// Mitsubishi GX Works2 project: traffic signal with data   PLC: FX1N/FX1NC

PROGRAM MAIN
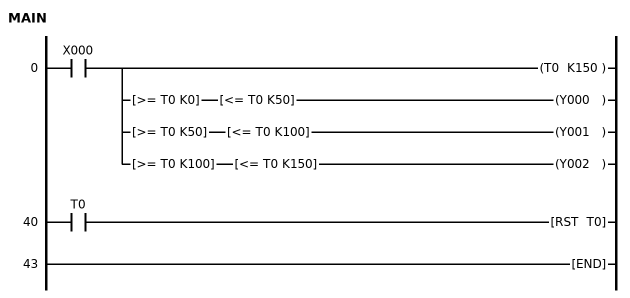
0     LD      X000
      OUT     T0 K150
      MPS
      AND>=   T0 K0
      AND<=   T0 K50
      OUT     Y000
      MRD
      AND>=   T0 K50
      AND<=   T0 K100
      OUT     Y001
      MPP
      AND>=   T0 K100
      AND<=   T0 K150
      OUT     Y002
40    LD      T0
      RST     T0
43    END
END_PROGRAM
